TYPE ST001_ProcessData EXTENDS TcoData.TcoEntity: 
STRUCT
END_STRUCT
END_TYPE

(* stored: Version 1.1.0.1, ProductVersion 3.1.4024.9
   DUT ST001_ProcessData: Id {eb62c574-36f6-0ac6-38b7-ede3c42ff585} *)
